(* IEC 61131-3 sources: Kur_TemplateProject_v1/TestPanelV1.fbsproj/MyController.device.xml.v3^/Plc Logic.plclogic.xml.v3^/Application.application.xml.v3^/Kur_Library/04_Programs, 1 file *)

(* ---- DateTime.prg.st ---- *)
PROGRAM DateTime
VAR
    RTCget      : DWORD;
    SetTime     : DWORD;
    pRes        : SysTimeRtc.RTS_IEC_RESULT;
    TimeLoaded  : BOOL;
END_VAR

// ---------- READ RTC ----------
SysTimeRtc.SysTimeRtcConvertUtcToDate(dwTimestampUtc := RTCget, pDate := Clock.Act);
SysTimeRtc.SysTimeRtcGet(pResult := pRes, SysTimeRtcGet => RTCget);

// ---------- LOAD CURRENT TIME INTO EDIT FIELDS ----------
IF TimeRead THEN
    Clock.Set  := Clock.Act;
    TimeRead   := FALSE;
    TimeLoaded := TRUE;
END_IF

// ---------- WRITE RTC ----------
IF TimeWrite AND TimeLoaded THEN
    SysTimeRtc.SysTimeRtcConvertDateToUtc(pDate := Clock.Set, pdwTimestampUtc := SetTime);
    SysTimeRtc.SysTimeRtcSet(ulTimestamp := SetTime);
    TimeWrite  := FALSE;
    TimeLoaded := FALSE;
END_IF
